FUNCTION_BLOCK FB_StepperMotor
VAR
    fbPower       : MC_Power;
	fbstop        : MC_Halt;
    fbMoveAbs     : MC_MoveAbsolute;
	fbhome		  : MC_Home;
    AxisRef       : AXIS_REF;
END_VAR

METHOD Enable : BOOL
VAR_INPUT
    bEnable : BOOL;
END_VAR
fbPower(Axis := AxisRef, Enable := bEnable);
Enable := NOT fbPower.Error;
END_METHOD

METHOD FB_init : BOOL
VAR_INPUT
    bInitRetains : BOOL;            // System-managed retains (not used here)
    bInCopyCode : BOOL;             // System-managed copy code (not used here)
    Axis        : AXIS_REF;         
END_VAR
 AxisRef := Axis;                
 FB_Init := TRUE;
END_METHOD

METHOD Home : BOOL
VAR_INPUT
    bExecute : BOOL;     
END_VAR

VAR
    bBusy    : BOOL;
    bDone    : BOOL;
    bError   : BOOL;
    nErrID   : UDINT;
END_VAR
fbHome(
    Execute       := bExecute,
	Axis		  := AxisRef,
	Position      := 0.0,       
    HomingMode    := 1,         
    Done          => bDone,
    Busy          => bBusy,
    Error         => bError,
    ErrorID       => nErrID
);

IF bDone THEN
    //Do something
ELSIF bError THEN
    //Do something
END_IF
END_METHOD

METHOD MoveToPosition : BOOL
VAR_INPUT
    fPosition : LREAL;
END_VAR
fbMoveAbs(Axis := AxisRef, Execute := TRUE, Position := fPosition);
MoveToPosition := NOT fbMoveAbs.Error;
END_METHOD

METHOD Stop : BOOL
VAR_INPUT
    bEnable : BOOL;
	bStopCommand : BOOL;
	fDecel : LREAL;
END_VAR
fbStop(Axis := AxisRef, Execute := bStopCommand, Deceleration := fDecel);
END_METHOD

END_FUNCTION_BLOCK

(* stored: Version 1.1.0.1, ProductVersion 3.1.4024.14
   POU FB_StepperMotor: Id {bbe3d249-0f45-4d4f-9e26-26a436162bb5}, SpecialFunc None
   Method Enable: Id {b4ed9b41-5152-4967-b132-962092157051}
   Method FB_init: Id {9d664a39-5dd4-4344-b1ab-aba2f4872a25}
   Method Home: Id {8276e0ce-98e0-421a-babf-511ef600c743}
   Method MoveToPosition: Id {59187d53-eaea-489c-80e7-2ef214427a40}
   Method Stop: Id {9b515f94-46a2-4ab1-aca0-af2dcdfe9f04} *)
